PROGRAM progLITCntrl
VAR
	LIT_04_0100 : fbLIT;
	
	LIT_04_1001 : fbLIT;
	LIT_04_1002 : fbLIT;
	LIT_04_1003 : fbLIT;

END_VAR

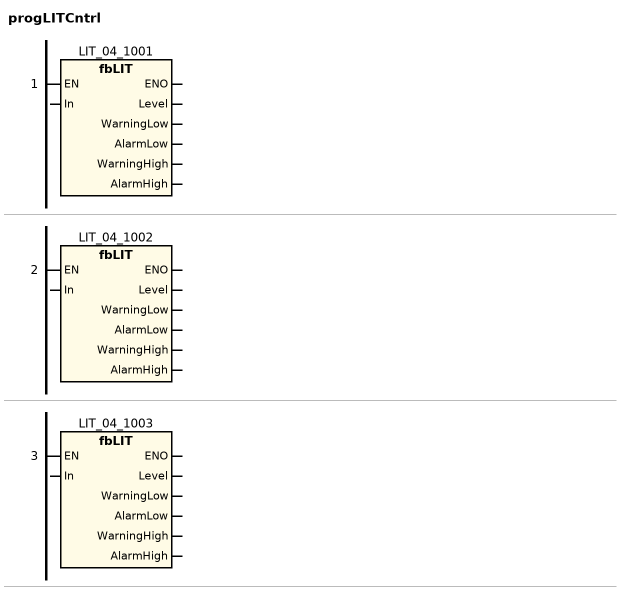
// NETWORK 1
LIT_04_1001(); // fbLIT

// NETWORK 2
LIT_04_1002(); // fbLIT

// NETWORK 3
LIT_04_1003(); // fbLIT

END_PROGRAM

(* stored: Version 1.1.0.1, ProductVersion 3.1.4022.17
   POU progLITCntrl: Id {8abdf04c-8ee3-442b-b85c-c2441be0b46a}, SpecialFunc None *)
